// TIA Portal V17 export
// export: Created 2025-03-10T13:12:10.530532Z, ExportSetting WithDefaults, DisplayName Totally Integrated Automation Portal, DisplayVersion V17 Update 8, DisplayName TIA Portal Openness, DisplayVersion V17 Update 8, DisplayName TIA Portal Version Control Interface, DisplayVersion V17, DisplayName SINAMICS Startdrive Advanced, DisplayVersion V17 SP2, DisplayName SINAMICS Startdrive G110M, G120, G120C, G120D, G120P, G115D, DisplayVersion V17 SP2, DisplayName SINAMICS Startdrive G130, G150, S120, S150, SINAMICS MV, S210, DisplayVersion V17 SP2, DisplayName STEP 7 Professional, DisplayVersion V17 Update 8, DisplayName SINUMERIK ONE STEP 7 Toolbox, DisplayVersion V17 Update 12, DisplayName SINUMERIK 840D sl STEP 7 Toolbox, DisplayVersion V17 Update 12, DisplayName STEP 7 Safety, DisplayVersion V17 Update 6, DisplayName WinCC Advanced, DisplayVersion V17 Update 8
TYPE "AUTO_SINGLE_SEMI_MANUAL"
// stored: IsFailsafeCompliant false
   STRUCT
      MANUAL_INPUT : Bool;   // MANUAL INPUT / MANUAL MODE INPUT
      SEMIAUTO_INPUT : Bool;   // SEMIAUTO INPUT / SEMIAUTOMATIC MODE INPUT
      AUTOMATIC_INPUT : Bool;   // AUTOMATIC INPUT / AUTOMATIC MODE INPUT
      SINGLE_INPUT : Bool;   // SINGLE CYCLE INPUT / SINGLE MODE INPUT
      NO_MODE_INPUT : Bool;   // NO MODE INPUT
      JOG_INPUT : Bool;   // JOG INPUT / JOG MODE INPUT
      TOOL_CHANGE_INPUT : Bool;   // TOOL CHANGE INPUT / TOOL CHANGE MODE INPUT
      CHANGE_GENERAL_CONDITIONS : Bool;   // CHANGE GENERAL CONDITIONS / CHANGE MODE GENERAL CONDITIONS
      CHANGE_INITIAL_CONDITIONS : Bool;   // CHANGE INITIAL CONDITIONS / CHANGE MODE INITIAL CONDITIONS
      MANUAL_REQUEST : Bool;   // MANUAL REQUEST / MANUAL MODE REQUEST
      SEMIAUTO_REQUEST : Bool;   // SEMIAUTO REQUEST / SEMIAUTOMATIC MODE REQUEST
      AUTOMATIC_REQUEST : Bool;   // AUTOMATIC REQUEST / AUTOMATIC MODE REQUEST
      SINGLE_REQUEST : Bool;   // SINGLE CYCLE REQUEST / SINGLE MODE REQUEST
      NO_MODE_REQUEST : Bool;   // NO MODE REQUEST
      NO_MODE_P_REQUEST_P : Bool;   // NO MODE REQUEST POSITIVE PULSE / NO MODE POSITIVE PULSE REQUEST
      NO_MODE_N_REQUEST_P : Bool;   // NO MODE REQUEST NEGATIVE PULSE / NO MODE NEGATIVE PULSE REQUEST
      JOG_REQUEST : Bool;   // JOG REQUEST / JOG MODE REQUEST
      TOOL_CHANGE_REQUEST : Bool;   // TOOL CHANGE REQUEST / TOOL CHANGE MODE REQUEST
      CHANGE_TO_MANUAL : Bool;   // CHANGE TO MANUAL MODE
      CHANGE_TO_MANUAL_P : Bool;   // CHANGE TO MANUAL PULSE / CHANGE TO MANUAL MODE PULSE
      CHANGE_TO_SEMIAUTO : Bool;   // CHANGE TO SEMIAUTO MODE / CHANGE TO SEMIAUTOMATIC MODE
      CHANGE_TO_AUTOMATIC : Bool;   // CHANGE TO AUTOMATIC MODE
      CHANGE_TO_SINGLE : Bool;   // CHANGE TO SINGLE CYCLE MODE / CHANGE TO SINGLE MODE
      CHANGE_TO_NO_MODE : Bool;   // CHANGE TO NO MODE
      CHANGE_TO_JOG_MODE : Bool;   // CHANGE TO JOG MODE
      CHANGE_TO_TOOL_CHG_MODE : Bool;   // CHANGE TO TOOL CHANGE MODE
      CHANGE_MODE_SEQ_RUN : Bool;   // CHANGE MODE SEQUENCE RUNNING
      MANUAL_SELECTED : Bool;   // MANUAL MODE SELECTED
      SEMIAUTO_SELECTED : Bool;   // SEMIAUTO MODE SELECTED / SEMIAUTOMATIC MODE SELECTED
      AUTOMATIC_SELECTED : Bool;   // AUTOMATIC MODE SELECTED
      SINGLE_SELECTED : Bool;   // SINGLE CYCLE MODE SELECTED / SINGLE MODE SELECTED
      NO_MODE_SELECTED : Bool;   // NO MODE MODE SELECTED / NO MODE SELECTED
      JOG_SELECTED : Bool;   // JOG MODE SELECTED
      TOOL_CHANGE_MODE_SELECTED : Bool;   // TOOL CHANGE MODE SELECTED
      AUTO_SINGLE_SEMI_SELECTED : Bool;   // AUTO / SEMIAUTO / SINGLE CYCLE MODE SELECTED / AUTO SINGLE SEMI MODE SELECTED
      MANUAL_SELECTED_MEMORY : Bool;   // MEMORY CHANGE MANUAL MODE / MANUAL MODE SELECTED MEMORY
      SEMI_SELECTED_MEMORY : Bool;   // MEMORY CHANGE MANUAL MODE / SEMI MODE SELECTED MEMORY
      AUTO_SELECTED_MEMORY : Bool;   // MEMORY CHANGE MANUAL MODE / AUTO MODE SELECTED MEMORY
      SINGLE_SELECTED_MEMORY : Bool;   // MEMORY CHANGE MANUAL MODE / SINGLE MODE SELECTED MEMORY
      JOG_SELECTED_MEMORY : Bool;   // MEMORY CHANGE JOG MODE / JOG MODE SELECTED MEMORY
      CHANGE_GENERAL_CONDITIONS_HELP : Bool;   // MODE CHANGE FAULT / CHANGE MODE GENERAL CONDITIONS HELP
      CHANGE_TO_MANUAL_ALARM : Bool;   // MANUAL MODE CHANGE FAULT / CHANGE TO MANUAL MODE ALARM
      CHANGE_TO_SEMIAUTO_ALARM : Bool;   // SEMIAUTO MODE CHANGE FAULT / CHANGE TO SEMIAUTO MODE ALARM
      CHANGE_TO_AUTO_ALARM : Bool;   // AUTOMATIC MODE CHANGE FAULT / CHANGE TO AUTO MODE ALARM
      CHANGE_TO_SINGLE_ALARM : Bool;   // SINGLE CYCLE MODE CHANGE FAULT / CHANGE TO SINGLE MODE ALARM
      CHANGE_TO_NO_MODE_ALARM : Bool;   // NO MODE CHANGE FAULT / CHANGE TO NO MODE ALARM
      CHANGE_TO_JOG_MODE_ALARM : Bool;   // JOG MODE CHANGE FAULT / CHANGE TO JOG MODE ALARM
      ELECTRONIC_HANDWEHELL_ACTIVE : Bool;   // ELECTRONIC HANDWEHELL ACTIVE
      OPTIONS : Struct
         SGM : Bool;   // SGM MACHINE
         GM : Bool;   // GM MACHINE
         FORD : Bool;   // FORD MACHINE
         ETXETAR : Bool;   // ETXETAR MACHINE
      END_STRUCT;
   END_STRUCT;
END_TYPE
